ABB RobotStudio station: Session3a.rspag

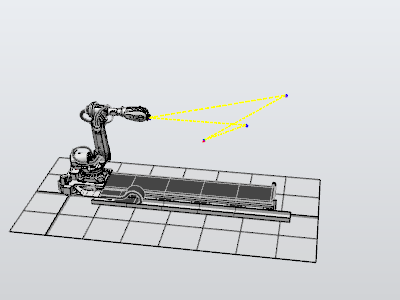
--- station ---
Station Station (saved by RobotStudio 24.2.10821.1)
Controller Controller3, task T_ROB1: task frame (RAPID world) sits at (590.5, 475, 384.5) mm in the station
Controller Controller3
  mechanical unit ROB_1: IRB6700_235_265_MH3_04, 6 joints, base frame (0, 0, 0) mm
  mechanical unit TRACK_1: IRBT6004_STD_0_0_5__04, 1 joints, base frame (0, 0, 0) mm
Layout (positions relative to the parent item):
  - IRB6700_235_265_MH3_04 [mechanism, from %ABB.RobotStudio.Models.IRB6700%\IRB6700_235_265_MH3_04.rslib] at (590.5, 475, 384.5) mm; joint values [0, 0, 0, 0, 0.5236, 0] (rad or m)
  - IRBT6004_STD_0_0_5__04 [mechanism] at (0, 0, 0) mm; joint values [0] (rad or m)
      links: Base, Link1
Attachment: IRB6700_235_265_MH3_04 is attached to IRBT6004_STD_0_0_5__04 / Link1

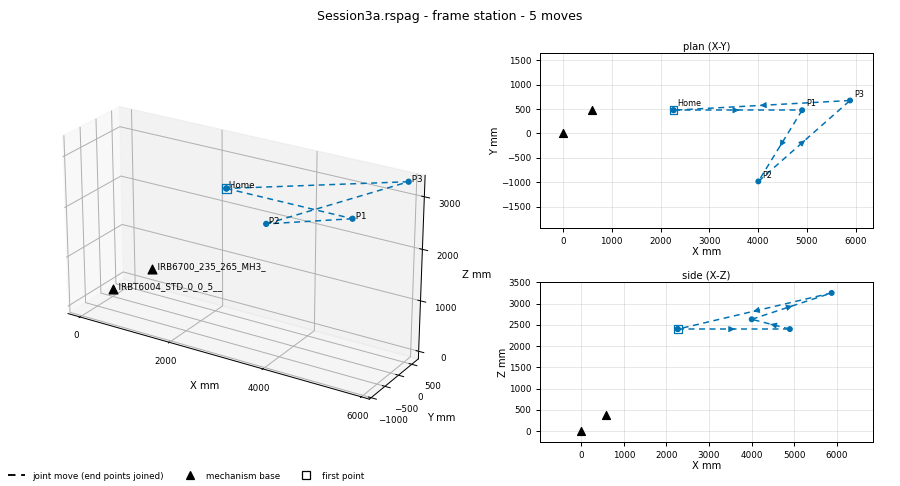
[picture p0: tool path of Session3a.rspag in frame station, 5 of 5 moves have a stored position in this frame; points joined in program order, loops and branches not executed]
--- Backups/Controller3/RAPID/TASK1/PROGMOD/Module1.mod ---
MODULE Module1
        CONST robtarget Home:=[[1675.705080757,0,2015],[0.5,0,0.866025404,0],[-1,0,-1,0],[0,9E+09,9E+09,9E+09,9E+09,9E+09]];
    CONST robtarget P1:=[[4310.280660193,0,2015],[0.5,0,0.866025404,0],[-1,0,-1,0],[2634.575579436,9E+09,9E+09,9E+09,9E+09,9E+09]];
    CONST robtarget P2:=[[3413.754627556,-1459.024830695,2245.511786952],[0.779589109,0.214342345,0.357460336,-0.467461537],[-1,-1,0,1],[2634.575579436,9E+09,9E+09,9E+09,9E+09,9E+09]];
    CONST robtarget P3:=[[5292.972895466,199.844942192,2864.679625378],[0.579383934,-0.071035248,0.810347417,0.051042273],[0,0,0,0],[4161.41039584,9E+09,9E+09,9E+09,9E+09,9E+09]];
!***********************************************************
    !
    ! Module:  Module1
    !
    ! Description:
    !   <Insert description here>
    !
    ! Author: ahmadk
    !
    ! Version: 1.0
    !
    !***********************************************************


    !***********************************************************
    !
    ! Procedure main
    !
    !   This is the entry point of your program
    !
    !***********************************************************
    PROC main()
        !Add your code here
        Path_10;
    ENDPROC
    PROC Path_10()
        MoveJ Home,v1500,z10,tool0\WObj:=wobj0;
        MoveJ P1,v1500,z10,tool0\WObj:=wobj0;
        MoveJ P2,v1500,z10,tool0\WObj:=wobj0;
        MoveJ P3,v1500,z10,tool0\WObj:=wobj0;
        MoveJ Home,v1500,z10,tool0\WObj:=wobj0;
    ENDPROC
ENDMODULE
